// TIA Portal project "SVETLOMET" (V20)

(* hardware
DEVICE "S7-1200 station_1"  S7-1200 Station
   slot 0: "Rack_0"  S7-1200 Rack  Rack  V1.0
   slot 1: "PLC_SVETLOMET"  CPU 1215C DC/DC/DC  6ES7 215-1AG40-0XB0  V4.7
*)

// ===== PLC "PLC_SVETLOMET"  CPU 1215C DC/DC/DC =====

VAR_GLOBAL   // PLC tag table "Default tag table"
   "Tag_1" AT %M0.0 : Bool;
   "Tag_2" AT %M0.1 : Bool;
   "Tag_3" AT %M0.2 : Bool;
   "Tag_4" AT %M0.3 : Bool;
   "Tag_5" AT %M0.4 : Bool;
   "Tag_6" AT %M0.5 : Bool;
END_VAR

DATA_BLOCK "prg_Svetlomet_SCL_DB"   // DB1
{ S7_Optimized_Access := 'TRUE' }
VERSION : 0.1
// stored: InstanceOfName prg_Svetlomet_SCL
"prg_Svetlomet_SCL"
BEGIN
END_DATA_BLOCK

FUNCTION_BLOCK "prg_Svetlomet_SCL"   // FB2, SCL
{ S7_Optimized_Access := 'TRUE' }
VERSION : 0.1
   VAR_INPUT
      START_TESTOVANI : Bool;   // Tlačítko START
      RESET : Bool;   // Tlačítko RESET
      CIDLO_POLOHY : Bool;   // Světlomet je správně usazen
      CIDLO_PRIPOJENI_KONEKTORU : Bool;   // Konektor připojen
      TESTER_RESPONSE : Bool;   // Výsledek testeru po dokončení celé sekvence
      TESTER_ERROR : Bool;   // Chyba / přerušení testu ze strany testeru
      CAS_OBRYSOVE : Time := T#3s;   // x
      POCET_BLIKNUTI : Int := 3;   // y
      CAS_BRZDOVE : Time := T#3s;   // z
   END_VAR
   VAR_OUTPUT
      OBRYSOVE_SVETLO : Bool;
      BLINKR : Bool;
      BRZDOVE_SVETLO : Bool;
      PRIPRAVENO : Bool;
      TEST_BEZI : Bool;
      HOTOVO : Bool;
      CHYBA_PODMINEK : Bool;
      CHYBA_TESTERU : Bool;
      KROK : Int;
      POCET_OTESTOVANYCH_SVETLOMETU : DInt;
      POCET_SPRAVNYCH_SVETLOMETU : DInt;
      POCET_CHYBNYCH_SVETLOMETU : DInt;
      POCET_DOKONCENYCH_TESTU : DInt;
   END_VAR
   VAR
      stav : Int := 0;
      ready : Bool;
      start_old : Bool;
      start_rise : Bool;
      chybaPodminekLatched : Bool;
      chybaTesteruLatched : Bool;
      blinkTarget : Int;
      blinkIndex : Int;
      vysledekZapsan : Bool;
      testerResponseSeenTrue : Bool;
      tonObrys : TON_TIME;
      tonBlinkOn : TON_TIME;
      tonBlinkOff : TON_TIME;
      tonBrzda : TON_TIME;
      tonVse : TON_TIME;
      tonTesterResponse : TON_TIME;
   END_VAR
BEGIN
   // ---------------------------------------------------------------------
   // Pomocné signály
   // ---------------------------------------------------------------------
   #ready := #CIDLO_POLOHY AND #CIDLO_PRIPOJENI_KONEKTORU;

   IF #POCET_BLIKNUTI < 1 THEN
       #blinkTarget := 1;
   ELSE
       #blinkTarget := #POCET_BLIKNUTI;
   END_IF;

   #start_rise := #START_TESTOVANI AND NOT #start_old;
   #start_old := #START_TESTOVANI;

   // ---------------------------------------------------------------------
   // RESET procesu (počítadla se nemažou)
   // ---------------------------------------------------------------------
   IF #RESET THEN
       #stav := 0;
       #chybaPodminekLatched := FALSE;
       #chybaTesteruLatched := FALSE;
       #blinkIndex := 0;
       #vysledekZapsan := FALSE;
       #testerResponseSeenTrue := FALSE;
   END_IF;

   // ---------------------------------------------------------------------
   // Ztráta základních podmínek během testu
   // ---------------------------------------------------------------------
   IF ((#stav >= 20) AND (#stav <= 55)) AND (NOT #ready) THEN
       #stav := 0;
       #chybaPodminekLatched := TRUE;
       #blinkIndex := 0;
       #vysledekZapsan := FALSE;
       #testerResponseSeenTrue := FALSE;
   END_IF;

   // ---------------------------------------------------------------------
   // Chyba ze strany testeru - okamžité ukončení jako NOK
   // ---------------------------------------------------------------------
   IF ((#stav >= 20) AND (#stav <= 55)) AND #TESTER_ERROR THEN
       #chybaTesteruLatched := TRUE;

       IF NOT #vysledekZapsan THEN
           #POCET_OTESTOVANYCH_SVETLOMETU := #POCET_OTESTOVANYCH_SVETLOMETU + 1;
           #POCET_CHYBNYCH_SVETLOMETU := #POCET_CHYBNYCH_SVETLOMETU + 1;
           #vysledekZapsan := TRUE;
       END_IF;

       #blinkIndex := 0;
       #testerResponseSeenTrue := FALSE;
       #stav := 70;
   END_IF;

   // ---------------------------------------------------------------------
   // Stavový automat
   // ---------------------------------------------------------------------
   CASE #stav OF

           // ==============================================================
           // 0 - IDLE
           // ==============================================================
       0:
           #OBRYSOVE_SVETLO := FALSE;
           #BLINKR := FALSE;
           #BRZDOVE_SVETLO := FALSE;

           #tonObrys(IN := FALSE,
                     PT := #CAS_OBRYSOVE);
           #tonBlinkOn(IN := FALSE,
                       PT := T#1s);
           #tonBlinkOff(IN := FALSE,
                        PT := T#1s);
           #tonBrzda(IN := FALSE,
                     PT := #CAS_BRZDOVE);
           #tonVse(IN := FALSE,
                   PT := T#5s);
           #tonTesterResponse(IN := FALSE,
                              PT := T#1s);

           IF #start_rise THEN
               IF #ready AND (NOT #TESTER_ERROR) THEN
                   #chybaPodminekLatched := FALSE;
                   #chybaTesteruLatched := FALSE;
                   #blinkIndex := 0;
                   #vysledekZapsan := FALSE;
                   #testerResponseSeenTrue := FALSE;
                   #stav := 20;
               ELSE
                   IF NOT #ready THEN
                       #chybaPodminekLatched := TRUE;
                   END_IF;

                   IF #TESTER_ERROR THEN
                       #chybaTesteruLatched := TRUE;
                   END_IF;
               END_IF;
           END_IF;

           // ==============================================================
           // 20 - OBRYSOVE
           // ==============================================================
       20:
           #OBRYSOVE_SVETLO := TRUE;
           #BLINKR := FALSE;
           #BRZDOVE_SVETLO := FALSE;

           #tonObrys(IN := TRUE,
                     PT := #CAS_OBRYSOVE);
           #tonBlinkOn(IN := FALSE,
                       PT := T#1s);
           #tonBlinkOff(IN := FALSE,
                        PT := T#1s);
           #tonBrzda(IN := FALSE,
                     PT := #CAS_BRZDOVE);
           #tonVse(IN := FALSE,
                   PT := T#5s);
           #tonTesterResponse(IN := FALSE,
                              PT := T#1s);

           IF #tonObrys.Q THEN
               #blinkIndex := 0;
               #stav := 30;
           END_IF;

           // ==============================================================
           // 30 - BLINKR ON
           // ==============================================================
       30:
           #OBRYSOVE_SVETLO := FALSE;
           #BLINKR := TRUE;
           #BRZDOVE_SVETLO := FALSE;

           #tonObrys(IN := FALSE,
                     PT := #CAS_OBRYSOVE);
           #tonBlinkOn(IN := TRUE,
                       PT := T#1s);
           #tonBlinkOff(IN := FALSE,
                        PT := T#1s);
           #tonBrzda(IN := FALSE,
                     PT := #CAS_BRZDOVE);
           #tonVse(IN := FALSE,
                   PT := T#5s);
           #tonTesterResponse(IN := FALSE,
                              PT := T#1s);

           IF #tonBlinkOn.Q THEN
               #stav := 31;
           END_IF;

           // ==============================================================
           // 31 - BLINKR OFF
           // ==============================================================
       31:
           #OBRYSOVE_SVETLO := FALSE;
           #BLINKR := FALSE;
           #BRZDOVE_SVETLO := FALSE;

           #tonObrys(IN := FALSE,
                     PT := #CAS_OBRYSOVE);
           #tonBlinkOn(IN := FALSE,
                       PT := T#1s);
           #tonBlinkOff(IN := TRUE,
                        PT := T#1s);
           #tonBrzda(IN := FALSE,
                     PT := #CAS_BRZDOVE);
           #tonVse(IN := FALSE,
                   PT := T#5s);
           #tonTesterResponse(IN := FALSE,
                              PT := T#1s);

           IF #tonBlinkOff.Q THEN
               #blinkIndex := #blinkIndex + 1;

               IF #blinkIndex < #blinkTarget THEN
                   #stav := 30;
               ELSE
                   #stav := 40;
               END_IF;
           END_IF;

           // ==============================================================
           // 40 - BRZDOVE
           // ==============================================================
       40:
           #OBRYSOVE_SVETLO := FALSE;
           #BLINKR := FALSE;
           #BRZDOVE_SVETLO := TRUE;

           #tonObrys(IN := FALSE,
                     PT := #CAS_OBRYSOVE);
           #tonBlinkOn(IN := FALSE,
                       PT := T#1s);
           #tonBlinkOff(IN := FALSE,
                        PT := T#1s);
           #tonBrzda(IN := TRUE,
                     PT := #CAS_BRZDOVE);
           #tonVse(IN := FALSE,
                   PT := T#5s);
           #tonTesterResponse(IN := FALSE,
                              PT := T#1s);

           IF #tonBrzda.Q THEN
               #stav := 50;
           END_IF;

           // ==============================================================
           // 50 - VSECHNA_SVETLA 5 s
           // ==============================================================
       50:
           #OBRYSOVE_SVETLO := TRUE;
           #BLINKR := TRUE;
           #BRZDOVE_SVETLO := TRUE;

           #tonObrys(IN := FALSE,
                     PT := #CAS_OBRYSOVE);
           #tonBlinkOn(IN := FALSE,
                       PT := T#1s);
           #tonBlinkOff(IN := FALSE,
                        PT := T#1s);
           #tonBrzda(IN := FALSE,
                     PT := #CAS_BRZDOVE);
           #tonVse(IN := TRUE,
                   PT := T#5s);
           #tonTesterResponse(IN := FALSE,
                              PT := T#1s);

           IF #tonVse.Q THEN
               #testerResponseSeenTrue := FALSE;
               #stav := 55;
           END_IF;

           // ==============================================================
           // 55 - 1 s čekání na TESTER_RESPONSE po úplném dokončení testu
           // ==============================================================
       55:
           #OBRYSOVE_SVETLO := FALSE;
           #BLINKR := FALSE;
           #BRZDOVE_SVETLO := FALSE;

           #tonObrys(IN := FALSE,
                     PT := #CAS_OBRYSOVE);
           #tonBlinkOn(IN := FALSE,
                       PT := T#1s);
           #tonBlinkOff(IN := FALSE,
                        PT := T#1s);
           #tonBrzda(IN := FALSE,
                     PT := #CAS_BRZDOVE);
           #tonVse(IN := FALSE,
                   PT := T#5s);
           #tonTesterResponse(IN := TRUE,
                              PT := T#1s);

           // Pokud se během této 1 s objeví TRUE, uloží se jako OK
           IF #TESTER_RESPONSE THEN
               #testerResponseSeenTrue := TRUE;
           END_IF;

           IF #tonTesterResponse.Q THEN
               IF NOT #vysledekZapsan THEN
                   #POCET_OTESTOVANYCH_SVETLOMETU := #POCET_OTESTOVANYCH_SVETLOMETU + 1;

                   IF #testerResponseSeenTrue THEN
                       #POCET_SPRAVNYCH_SVETLOMETU := #POCET_SPRAVNYCH_SVETLOMETU + 1;
                   ELSE
                       #POCET_CHYBNYCH_SVETLOMETU := #POCET_CHYBNYCH_SVETLOMETU + 1;
                   END_IF;

                   #vysledekZapsan := TRUE;
               END_IF;

               #POCET_DOKONCENYCH_TESTU := #POCET_DOKONCENYCH_TESTU + 1;
               #stav := 60;
           END_IF;

           // ==============================================================
           // 60 - HOTOVO
           // ==============================================================
       60:
           #OBRYSOVE_SVETLO := FALSE;
           #BLINKR := FALSE;
           #BRZDOVE_SVETLO := FALSE;

           #tonObrys(IN := FALSE,
                     PT := #CAS_OBRYSOVE);
           #tonBlinkOn(IN := FALSE,
                       PT := T#1s);
           #tonBlinkOff(IN := FALSE,
                        PT := T#1s);
           #tonBrzda(IN := FALSE,
                     PT := #CAS_BRZDOVE);
           #tonVse(IN := FALSE,
                   PT := T#5s);
           #tonTesterResponse(IN := FALSE,
                              PT := T#1s);

           IF #start_rise THEN
               IF #ready AND (NOT #TESTER_ERROR) THEN
                   #chybaPodminekLatched := FALSE;
                   #chybaTesteruLatched := FALSE;
                   #blinkIndex := 0;
                   #vysledekZapsan := FALSE;
                   #testerResponseSeenTrue := FALSE;
                   #stav := 20;
               ELSE
                   IF NOT #ready THEN
                       #chybaPodminekLatched := TRUE;
                   END_IF;

                   IF #TESTER_ERROR THEN
                       #chybaTesteruLatched := TRUE;
                   END_IF;
               END_IF;
           END_IF;

           // ==============================================================
           // 70 - CHYBA TESTERU
           // ==============================================================
       70:
           #OBRYSOVE_SVETLO := FALSE;
           #BLINKR := FALSE;
           #BRZDOVE_SVETLO := FALSE;

           #tonObrys(IN := FALSE,
                     PT := #CAS_OBRYSOVE);
           #tonBlinkOn(IN := FALSE,
                       PT := T#1s);
           #tonBlinkOff(IN := FALSE,
                        PT := T#1s);
           #tonBrzda(IN := FALSE,
                     PT := #CAS_BRZDOVE);
           #tonVse(IN := FALSE,
                   PT := T#5s);
           #tonTesterResponse(IN := FALSE,
                              PT := T#1s);

           IF #start_rise THEN
               IF #ready AND (NOT #TESTER_ERROR) THEN
                   #chybaPodminekLatched := FALSE;
                   #chybaTesteruLatched := FALSE;
                   #blinkIndex := 0;
                   #vysledekZapsan := FALSE;
                   #testerResponseSeenTrue := FALSE;
                   #stav := 20;
               ELSE
                   IF NOT #ready THEN
                       #chybaPodminekLatched := TRUE;
                   END_IF;

                   IF #TESTER_ERROR THEN
                       #chybaTesteruLatched := TRUE;
                   END_IF;
               END_IF;
           END_IF;

       ELSE
           #stav := 0;

   END_CASE;

   // ---------------------------------------------------------------------
   // Stavové výstupy
   // ---------------------------------------------------------------------
   #TEST_BEZI := (#stav >= 20) AND (#stav <= 55);
   #PRIPRAVENO := #ready AND (NOT #TESTER_ERROR) AND ((#stav = 0) OR (#stav = 60) OR (#stav = 70));
   #HOTOVO := (#stav = 60);
   #CHYBA_PODMINEK := #chybaPodminekLatched;
   #CHYBA_TESTERU := #chybaTesteruLatched;
   #KROK := #stav;
END_FUNCTION_BLOCK

ORGANIZATION_BLOCK "Main"   // OB1, LAD, ProgramCycle
TITLE = "Main Program Sweep (Cycle)"
{ S7_Optimized_Access := 'TRUE' }
VERSION : 0.1
   VAR_INPUT
      Initial_Call : Bool;   // Initial call of this OB
      Remanence : Bool;   // =True, if remanent data are available
   END_VAR
BEGIN

REGION Network 1
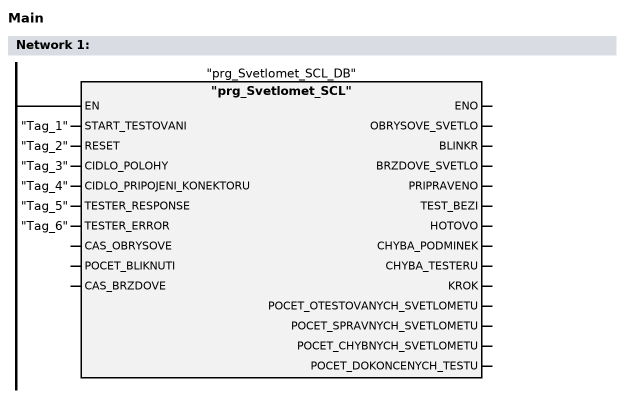
   RUNG wire#powerrail
      "prg_Svetlomet_SCL_DB"(START_TESTOVANI := "Tag_1", RESET := "Tag_2", CIDLO_POLOHY := "Tag_3", CIDLO_PRIPOJENI_KONEKTORU := "Tag_4", CAS_OBRYSOVE :=, POCET_BLIKNUTI :=, CAS_BRZDOVE :=, TESTER_RESPONSE := "Tag_5", TESTER_ERROR := "Tag_6", OBRYSOVE_SVETLO =>, BLINKR =>, BRZDOVE_SVETLO =>, PRIPRAVENO =>, TEST_BEZI =>, HOTOVO =>, CHYBA_PODMINEK =>, CHYBA_TESTERU =>, KROK =>, POCET_DOKONCENYCH_TESTU =>, POCET_OTESTOVANYCH_SVETLOMETU =>, POCET_SPRAVNYCH_SVETLOMETU =>, POCET_CHYBNYCH_SVETLOMETU =>)
   END_RUNG
   // the same network as SCL:
   "prg_Svetlomet_SCL_DB"(START_TESTOVANI := "Tag_1",   // "prg_Svetlomet_SCL"
                          RESET := "Tag_2",
                          CIDLO_POLOHY := "Tag_3",
                          CIDLO_PRIPOJENI_KONEKTORU := "Tag_4",
                          TESTER_RESPONSE := "Tag_5",
                          TESTER_ERROR := "Tag_6");
END_REGION
END_ORGANIZATION_BLOCK